FUNCTION_BLOCK Test_AssertEquals_DWORD EXTENDS T_UnitTestBase
VAR
    AssertionUnderTest : T_Assertion(AssertionListenerMock);
    AssertionListenerMock : T_AssertionListenerMock;
    DWORD_Variable : DWORD;
END_VAR

// Initialise the classes under test (may be repaeting the tests)...
AssertionListenerMock.fb_Init(
    bInitRetains      := FALSE,
	bInCopyCode       := FALSE);
AssertionUnderTest.fb_Init(
    bInitRetains      := FALSE,
	bInCopyCode       := FALSE,
    AssertionListener := AssertionListenerMock);

// Test the assertion...
DWORD_Variable := 1111;

AssertionUnderTest.AssertEquals_DWORD(
    Expected := 2222, // deliberately different to test the assertion
    Actual   := DWORD_Variable,
    VariableName := 'DWORD_Variable');
 
    
// Check the assertion worked...    
Assertion.AssertEquals_BOOL(
    Expected := TRUE,
    Actual   := AssertionListenerMock.AssertionFailed,
    VariableName := 'AssertionListenerMock.AssertionFailed');

// Check the assertion messages...    
Assertion.AssertEquals_STRING(
    Expected := 'AssertEquals_DWORD failed in AssertionListenerMock: Value "DWORD_Variable"',
    Actual   := AssertionListenerMock.AssertionMessage,
    VariableName := 'AssertionListenerMock.AssertionMessage');

Assertion.AssertEquals_STRING(
    Expected := '  Expected = 2222',
    Actual   := AssertionListenerMock.ExpectedAsString,
    VariableName := 'AssertionListenerMock.ExpectedAsString');

Assertion.AssertEquals_STRING(
    Expected := '  Actual   = 1111',
    Actual   := AssertionListenerMock.ActualAsString,
    VariableName := 'AssertionListenerMock.ActualAsString');

TestFinished();

END_FUNCTION_BLOCK

(* stored: Version 1.1.0.1, ProductVersion 3.1.4024.4
   POU Test_AssertEquals_DWORD: Id {74850fe4-9dcb-406d-ab1e-3b2dbbcb5237}, SpecialFunc None *)
